VAR_GLOBAL
	//
	Start 			: BOOL;
	Reset 			: BOOL;
	Stop  			: BOOL;
	//
	StartLight		: BOOL;
	ResetLight		: BOOL;
	StopLight		: BOOL;
	//
	LevelMeter 		: INT;
	FlowMeter		: INT;
	SetPoint		: INT;
	//
	FillValve		: INT;
	DischargeValve	: INT;
	SP				: INT;
	PV				: INT;
	//
END_VAR

(* stored: Version 1.1.0.1, ProductVersion 3.1.4024.6
   GVL GlobalTags: Id {66cb291c-2657-471d-8555-fecf4d93ea15} *)
